// TwinCAT 3 PLC project Anker_Walfischgasse
// ProgramVersion: 3.1.4023.0
// libraries:
//   EfficientIO Communicator, * (EfficientIO)
//   EfficientIO Energy Basic, * (EfficientIO)
//   Lynus Persistent Data V1, * (Lynus AG)
//   Lynus Standards, * (EfficientIO)
//   Tc2_BABasic, * (Beckhoff Automation GmbH)
//   Tc2_Standard, * (Beckhoff Automation GmbH)
//   Tc2_System, * (Beckhoff Automation GmbH)
//   Tc2_Utilities, * (Beckhoff Automation GmbH)
//   Tc3_IotBase, * (Beckhoff Automation GmbH)
//   Tc3_JsonXml, * (Beckhoff Automation GmbH)
//   Tc3_Module, * (Beckhoff Automation GmbH)
// project tree:
//   / FastTask.TcTTO (not stored), MiddleTask.TcTTO, SlowTask.TcTTO (not stored)
//   FBs/ FB_Shelly_Pro1PM.TcPOU (not stored), FB_Shelly_Pro1PM_Helper.TcPOU, FB_TimeSwitch.TcPOU (not stored), FB_TimeSwitch_V2.TcPOU (not stored)
//   POUs/ prg5530Con.TcPOU, prg5530EMS.TcPOU, prgComEffIO.TcPOU, prg5530Grid.TcPOU (not stored), prgPersistent.TcPOU, prgRWEffIO.TcPOU (not stored), prgVarEffIO.TcPOU (not stored), prg_SystemTime.TcPOU (not stored)
// real-time tasks:
//   TASK FastTask: cycle T#5ms, priority 4, ADS port 350
//   TASK MiddleTask: cycle T#10ms, priority 8, ADS port 351
//   TASK SlowTask: cycle T#20ms, priority 10, ADS port 352
// I/O:
//   DEVICE Gerät 1 (Beckhoff CCAT)
//   DEVICE Gerät 2 (EtherCAT), AmsNetId 5.100.32.125.3.1
//     Klemme 1 (EK1200) [EK1200-5000 EtherCAT Netzteil (2A E-Bus)]
//       Klemme 2 (EL3443) [EL3443 3K. Leistungsmessung]
//       Klemme 3 (EL2652) [EL2652 2K. Relais Ausgang, Wechsler (230V AC / 30V DC)]
//       Klemme 4 (EL2652) [EL2652 2K. Relais Ausgang, Wechsler (230V AC / 30V DC)]
//       Klemme 5 (EL2652) [EL2652 2K. Relais Ausgang, Wechsler (230V AC / 30V DC)]
//       Klemme 6 (EL2652) [EL2652 2K. Relais Ausgang, Wechsler (230V AC / 30V DC)]
//       Klemme 7 (EL9011) [EL9011 Endklemme]

CONFIGURATION Anker_Walfischgasse
    RESOURCE PLC ON TwinCAT3
        TASK MiddleTask(INTERVAL := T#10ms, PRIORITY := 8);
        PROGRAM prgPersistent WITH MiddleTask : prgPersistent;
    END_RESOURCE
END_CONFIGURATION

// ---- POUs/prgPersistent.TcPOU
PROGRAM prgPersistent
VAR
	fbUSV		: FB_WritePersistentData_CX81xx;
	fb_Reboot		: NT_reboot;
	m_Reboot		: BOOL:=FALSE;
END_VAR

fbUSV(
	eSaveModeData:= eUSVSaveMode.eSaveWhenPowerfail, 
	bLoadPersistentDataOk=> , 
	bPowerFailDetect=> , 
	bError=> , 
	bySaveProcess=> , 
	dwStorageLast24h=> , 
	udiErrorCode=> );
	
prg_SystemTime();

		
fb_Reboot(	netid := '',
			delay := 2,
			start := m_Reboot);

END_PROGRAM

// ---- FBs/FB_Shelly_Pro1PM_Helper.TcPOU
FUNCTION_BLOCK FB_Shelly_Pro1PM_Helper
VAR_INPUT
	bSend			: BOOL;
	bSetOnP1		: BOOL;
	bSetOffP1		: BOOL;
END_VAR

VAR_IN_OUT
	fbClient		: FB_IotHttpClient;
END_VAR

VAR_OUTPUT
	bBusy			: BOOL;
	bError			: BOOL;
	bStateP1		: BOOL;
	lrapowerP1		: LREAL;
	lrvoltageP1		: LREAL;
	lraenergyP1		: LREAL;
	lrTemperatureP1	: LREAL;
END_VAR

VAR
	fbRequestSwitch0	: FB_IotHttpRequest;
	fbRequestSwitch1	: FB_IotHttpRequest;
	RisingEdge			: R_TRIG;
	RisingEdgeSetOnP1	: R_TRIG;
	RisingEdgeSetOffP1	: R_TRIG;
	fbJson				: FB_JsonDomParser;
	nState				: UDINT;
	timTimeout			: TON;
	tTimeOut			: TIME := T#2S;
	timTimeoutSwitch	: TON;
	tTimeOutSwitch		: TIME := T#5S;
	bGetContentResult	: BOOL;
	sContentS0			: STRING(511);
	
	bGetJsonResult		: BOOL;
	jsonDoc				: SJsonValue;
	jsonVal				: SJsonValue;
	
	nReqCount			: UDINT;	
	nResCount			: UDINT;
	nValidResCount		: UDINT;
	nErrCount			: UDINT;
	
	fbRequest2         : FB_IotHttpRequest;
	fbRequest3         : FB_IotHttpRequest;
	fbHeader            : FB_IotHttpHeaderFieldMap;
	fbHeader2            : FB_IotHttpHeaderFieldMap;
	
	sRealm	:	STRING(511);
	sPassword :	STRING(511) := ':sh3lly4ankerio2$$';
	snonce	:	STRING(511);
	scnonce	:	STRING(511);
	shash	: STRING(511);
	bhash	: BOOL;
	
	aData	: STRING(511);
	a_ha1	: ARRAY[0..31] OF BYTE;
	str_ha1 : STRING(511);
	str_Toha1   : STRING(511);
	udint_length_string : UDINT;
	
	a_ha2	: ARRAY[0..31] OF BYTE;
	str_ha2 : STRING(511);
	str_Toha2   : STRING(511);
	
	a_response	: ARRAY[0..31] OF BYTE;
	str_response : STRING(511);
	str_Toresponse   : STRING(511);

	str_authorization	: STRING(2048);
	
	sfincontent	: STRING(511);
	int_CountOffWrite: INT;
	int_CountOnWrite: INT;
	str_URI : STRING(50);
	int_Mode: INT;
	ton_Timeout: Ton;
	b_Done: BOOL;
	nState_Old: UDINT;
	int_ErrorCount: INT;
END_VAR

//Timer for Timeout
timTimeout(IN:= (nState = 1 AND bBusy) OR (nState = nState_Old AND bBusy), PT:= tTimeOut, Q=> , ET=> );
	IF timTimeout.Q THEN 
		nState := 0;
		bBusy := FALSE;
		bStateP1 := FALSE;
		lrapowerP1 := 0;
		lrvoltageP1 := 0;
		lraenergyP1 := 0;
		lrTemperatureP1 := 0;		
	END_IF
IF nState<> nState_old THEN
	nState_old := nState;
END_IF	
(*timTimeoutSwitch(IN:= bSetOnP1 OR bSetOffP1, PT:= tTimeOut, Q=> , ET=> );
	IF timTimeoutSwitch.Q THEN 
		bSetOnP1 := FALSE;
		bSetOffP1 := FALSE;
	END_IF
*)
IF bError THEN
	int_ErrorCount := int_ErrorCount+1;
	bError := FALSE;
END_IF

RisingEdge(CLK:= bSend );
RisingEdgeSetOnP1(CLK:= bSetOnP1 );
RisingEdgeSetOffP1(CLK:= bSetOffP1 );

CASE nState OF
	0:	
		IF RisingEdge.Q THEN 
			IF bSetOnP1 AND NOT b_Done THEN 
				// switch on
				str_URI :='/rpc/Switch.Set?id=0&on=true';
				int_Mode := 1;
				b_Done := TRUE;
				bBusy:= TRUE;
				bError:= FALSE;
				nState:= 1;
			ELSIF bSetOffP1 AND NOT b_Done THEN
				// switch off
				str_URI :='/rpc/Switch.Set?id=0&on=false';
				int_Mode := 2;
				b_Done := TRUE;
				bBusy:= TRUE;
				bError:= FALSE;
				nState:= 1;
			ELSIF ((bSetOnP1 OR bSetOffP1) AND  b_Done) OR (NOT bSetOnP1 AND NOT bSetOffP1) THEN
				// read
				str_URI :='/rpc/Switch.GetStatus?id=0';
				int_Mode := 0;
				b_Done := FALSE;
				bBusy:= TRUE;
				bError:= FALSE;
				nState:= 1;
			END_IF
		END_IF
	1:
		IF
			fbRequestSwitch0.SendRequest(sUri:=str_URI, fbClient:=fbClient, eRequestType:=ETcIotHttpRequestType.HTTP_Get, 0, 0, 0) THEN
			nState:= 2;
			nReqCount:= nReqCount+1;
		END_IF
	
	2:
		IF NOT fbRequestSwitch0.bBusy THEN
			bError:= TRUE;
			IF NOT fbRequestSwitch0.bError THEN
				bGetContentResult:= fbRequestSwitch0.GetHeaderField(pValue:= ADR(sContentS0), 
														 nValueSize:= SIZEOF(sContentS0), sField := 'WWW-Authenticate');
				IF fbRequestSwitch0.nStatusCode = 401 THEN
					bGetJsonResult:= FALSE;
						sRealm := sContentS0;
						sRealm := DELETE(sRealm, FIND(sRealm, 'realm') + 7, 0);
						sRealm := DELETE(sRealm, LEN(sRealm), FIND(sRealm, '"'));
						
						snonce := sContentS0;
						snonce := DELETE(snonce, FIND(snonce, 'nonce') + 7, 0);
						snonce := DELETE(snonce, LEN(snonce), FIND(snonce, '"'));
						
						scnonce := 'YmawvYzT';
					
						aData := sRealm;
						
						str_Toha1:=concat('admin:', sRealm);
						str_Toha1:=concat(str_Toha1, sPassword);
		 
						udint_length_string:= len2(ADR(str_Toha1));
						F_GenerateHashValue(E_HashMode.HASH_SHA256,ADR(str_Toha1),udint_length_string,ADR(a_ha1),32);
						
							str_ha1:=concat(byte_to_hexstr(a_ha1[0],2,TRUE),byte_to_hexstr(a_ha1[1],2,TRUE));
							str_ha1:=concat(str_ha1,byte_to_hexstr(a_ha1[2],2,TRUE));
							str_ha1:=concat(str_ha1,byte_to_hexstr(a_ha1[3],2,TRUE));
							str_ha1:=concat(str_ha1,byte_to_hexstr(a_ha1[4],2,TRUE));
							str_ha1:=concat(str_ha1,byte_to_hexstr(a_ha1[5],2,TRUE));
							str_ha1:=concat(str_ha1,byte_to_hexstr(a_ha1[6],2,TRUE));
							str_ha1:=concat(str_ha1,byte_to_hexstr(a_ha1[7],2,TRUE));
							str_ha1:=concat(str_ha1,byte_to_hexstr(a_ha1[8],2,TRUE));
							str_ha1:=concat(str_ha1,byte_to_hexstr(a_ha1[9],2,TRUE));
							str_ha1:=concat(str_ha1,byte_to_hexstr(a_ha1[10],2,TRUE));
							str_ha1:=concat(str_ha1,byte_to_hexstr(a_ha1[11],2,TRUE));
							str_ha1:=concat(str_ha1,byte_to_hexstr(a_ha1[12],2,TRUE));
							str_ha1:=concat(str_ha1,byte_to_hexstr(a_ha1[13],2,TRUE));
							str_ha1:=concat(str_ha1,byte_to_hexstr(a_ha1[14],2,TRUE));
							str_ha1:=concat(str_ha1,byte_to_hexstr(a_ha1[15],2,TRUE));
							str_ha1:=concat(str_ha1,byte_to_hexstr(a_ha1[16],2,TRUE));
							str_ha1:=concat(str_ha1,byte_to_hexstr(a_ha1[17],2,TRUE));
							str_ha1:=concat(str_ha1,byte_to_hexstr(a_ha1[18],2,TRUE));
							str_ha1:=concat(str_ha1,byte_to_hexstr(a_ha1[19],2,TRUE));
							str_ha1:=concat(str_ha1,byte_to_hexstr(a_ha1[20],2,TRUE));
							str_ha1:=concat(str_ha1,byte_to_hexstr(a_ha1[21],2,TRUE));
							str_ha1:=concat(str_ha1,byte_to_hexstr(a_ha1[22],2,TRUE));
							str_ha1:=concat(str_ha1,byte_to_hexstr(a_ha1[23],2,TRUE));
							str_ha1:=concat(str_ha1,byte_to_hexstr(a_ha1[24],2,TRUE));
							str_ha1:=concat(str_ha1,byte_to_hexstr(a_ha1[25],2,TRUE));
							str_ha1:=concat(str_ha1,byte_to_hexstr(a_ha1[26],2,TRUE));
							str_ha1:=concat(str_ha1,byte_to_hexstr(a_ha1[27],2,TRUE));
							str_ha1:=concat(str_ha1,byte_to_hexstr(a_ha1[28],2,TRUE));
							str_ha1:=concat(str_ha1,byte_to_hexstr(a_ha1[29],2,TRUE));
							str_ha1:=concat(str_ha1,byte_to_hexstr(a_ha1[30],2,TRUE));
							str_ha1:=concat(str_ha1,byte_to_hexstr(a_ha1[31],2,TRUE));
						
						str_Toha2:= concat('GET:',str_URI);
				 
						udint_length_string:= len2(ADR(str_Toha2));
						F_GenerateHashValue(E_HashMode.HASH_SHA256,ADR(str_Toha2),udint_length_string,ADR(a_ha2),32);
						
							str_ha2:=concat(byte_to_hexstr(a_ha2[0],2,TRUE),byte_to_hexstr(a_ha2[1],2,TRUE));
							str_ha2:=concat(str_ha2,byte_to_hexstr(a_ha2[2],2,TRUE));
							str_ha2:=concat(str_ha2,byte_to_hexstr(a_ha2[3],2,TRUE));
							str_ha2:=concat(str_ha2,byte_to_hexstr(a_ha2[4],2,TRUE));
							str_ha2:=concat(str_ha2,byte_to_hexstr(a_ha2[5],2,TRUE));
							str_ha2:=concat(str_ha2,byte_to_hexstr(a_ha2[6],2,TRUE));
							str_ha2:=concat(str_ha2,byte_to_hexstr(a_ha2[7],2,TRUE));
							str_ha2:=concat(str_ha2,byte_to_hexstr(a_ha2[8],2,TRUE));
							str_ha2:=concat(str_ha2,byte_to_hexstr(a_ha2[9],2,TRUE));
							str_ha2:=concat(str_ha2,byte_to_hexstr(a_ha2[10],2,TRUE));
							str_ha2:=concat(str_ha2,byte_to_hexstr(a_ha2[11],2,TRUE));
							str_ha2:=concat(str_ha2,byte_to_hexstr(a_ha2[12],2,TRUE));
							str_ha2:=concat(str_ha2,byte_to_hexstr(a_ha2[13],2,TRUE));
							str_ha2:=concat(str_ha2,byte_to_hexstr(a_ha2[14],2,TRUE));
							str_ha2:=concat(str_ha2,byte_to_hexstr(a_ha2[15],2,TRUE));
							str_ha2:=concat(str_ha2,byte_to_hexstr(a_ha2[16],2,TRUE));
							str_ha2:=concat(str_ha2,byte_to_hexstr(a_ha2[17],2,TRUE));
							str_ha2:=concat(str_ha2,byte_to_hexstr(a_ha2[18],2,TRUE));
							str_ha2:=concat(str_ha2,byte_to_hexstr(a_ha2[19],2,TRUE));
							str_ha2:=concat(str_ha2,byte_to_hexstr(a_ha2[20],2,TRUE));
							str_ha2:=concat(str_ha2,byte_to_hexstr(a_ha2[21],2,TRUE));
							str_ha2:=concat(str_ha2,byte_to_hexstr(a_ha2[22],2,TRUE));
							str_ha2:=concat(str_ha2,byte_to_hexstr(a_ha2[23],2,TRUE));
							str_ha2:=concat(str_ha2,byte_to_hexstr(a_ha2[24],2,TRUE));
							str_ha2:=concat(str_ha2,byte_to_hexstr(a_ha2[25],2,TRUE));
							str_ha2:=concat(str_ha2,byte_to_hexstr(a_ha2[26],2,TRUE));
							str_ha2:=concat(str_ha2,byte_to_hexstr(a_ha2[27],2,TRUE));
							str_ha2:=concat(str_ha2,byte_to_hexstr(a_ha2[28],2,TRUE));
							str_ha2:=concat(str_ha2,byte_to_hexstr(a_ha2[29],2,TRUE));
							str_ha2:=concat(str_ha2,byte_to_hexstr(a_ha2[30],2,TRUE));
							str_ha2:=concat(str_ha2,byte_to_hexstr(a_ha2[31],2,TRUE));
							
						// <ha1> + ":" + <nonce> + ":" + <nc> + ":" + <cnonce> + ":" + "auth" + ":" + <ha2>
						
						str_Toresponse:=concat(str_ha1,':');
						str_Toresponse:=concat(str_Toresponse,snonce);
						str_Toresponse:=concat(str_Toresponse,':00000001:');
						str_Toresponse:=concat(str_Toresponse,scnonce);
						str_Toresponse:=concat(str_Toresponse,':');
						str_Toresponse:=concat(str_Toresponse,'auth:');
						str_Toresponse:=concat(str_Toresponse,str_ha2);
						
						udint_length_string:= len2(ADR(str_Toresponse));
						F_GenerateHashValue(E_HashMode.HASH_SHA256,ADR(str_Toresponse),udint_length_string,ADR(a_response),32);
						
							str_response:=concat(byte_to_hexstr(a_response[0],2,TRUE),byte_to_hexstr(a_response[1],2,TRUE));
							str_response:=concat(str_response,byte_to_hexstr(a_response[2],2,TRUE));
							str_response:=concat(str_response,byte_to_hexstr(a_response[3],2,TRUE));
							str_response:=concat(str_response,byte_to_hexstr(a_response[4],2,TRUE));
							str_response:=concat(str_response,byte_to_hexstr(a_response[5],2,TRUE));
							str_response:=concat(str_response,byte_to_hexstr(a_response[6],2,TRUE));
							str_response:=concat(str_response,byte_to_hexstr(a_response[7],2,TRUE));
							str_response:=concat(str_response,byte_to_hexstr(a_response[8],2,TRUE));
							str_response:=concat(str_response,byte_to_hexstr(a_response[9],2,TRUE));
							str_response:=concat(str_response,byte_to_hexstr(a_response[10],2,TRUE));
							str_response:=concat(str_response,byte_to_hexstr(a_response[11],2,TRUE));
							str_response:=concat(str_response,byte_to_hexstr(a_response[12],2,TRUE));
							str_response:=concat(str_response,byte_to_hexstr(a_response[13],2,TRUE));
							str_response:=concat(str_response,byte_to_hexstr(a_response[14],2,TRUE));
							str_response:=concat(str_response,byte_to_hexstr(a_response[15],2,TRUE));
							str_response:=concat(str_response,byte_to_hexstr(a_response[16],2,TRUE));
							str_response:=concat(str_response,byte_to_hexstr(a_response[17],2,TRUE));
							str_response:=concat(str_response,byte_to_hexstr(a_response[18],2,TRUE));
							str_response:=concat(str_response,byte_to_hexstr(a_response[19],2,TRUE));
							str_response:=concat(str_response,byte_to_hexstr(a_response[20],2,TRUE));
							str_response:=concat(str_response,byte_to_hexstr(a_response[21],2,TRUE));
							str_response:=concat(str_response,byte_to_hexstr(a_response[22],2,TRUE));
							str_response:=concat(str_response,byte_to_hexstr(a_response[23],2,TRUE));
							str_response:=concat(str_response,byte_to_hexstr(a_response[24],2,TRUE));
							str_response:=concat(str_response,byte_to_hexstr(a_response[25],2,TRUE));
							str_response:=concat(str_response,byte_to_hexstr(a_response[26],2,TRUE));
							str_response:=concat(str_response,byte_to_hexstr(a_response[27],2,TRUE));
							str_response:=concat(str_response,byte_to_hexstr(a_response[28],2,TRUE));
							str_response:=concat(str_response,byte_to_hexstr(a_response[29],2,TRUE));
							str_response:=concat(str_response,byte_to_hexstr(a_response[30],2,TRUE));
							str_response:=concat(str_response,byte_to_hexstr(a_response[31],2,TRUE));
							
						// "Digest username=\"admin\", realm=\"shellypro4pm-083af27cfbac\", nonce=\"63768368\", uri=\"/rpc/Switch.GetStatus?id=0\", algorithm=\"SHA-256\", qop=auth, nc=00000001, cnonce=\"oKOklSrS\", response=\"d1d59d1e015dee0a3acfc97b20a0fa0ff851b03d79ca00df59ce018a63041468\""
						
						str_authorization:=concat('Digest username="admin", realm="',sRealm);
						str_authorization:=concat(str_authorization,'", nonce="');
						str_authorization:=concat(str_authorization,snonce);
						str_authorization:=concat(str_authorization,'", algorithm="SHA-256", uri="');
						str_authorization:=concat(str_authorization,str_URI);
						str_authorization:=concat(str_authorization,'", qop=auth, nc=00000001, cnonce="');
						str_authorization:=concat(str_authorization,scnonce);
						str_authorization:=concat(str_authorization,'", response="');
						str_authorization:=concat(str_authorization,str_response);
						str_authorization:=concat(str_authorization,'"');
						
						fbHeader.AddField('Authorization', str_authorization, FALSE);
						IF fbRequest2.SendRequest(sUri:= str_URI, fbClient:= fbClient, eRequestType:= ETcIotHttpRequestType.HTTP_Get, 0, 0, fbHeader) THEN
							nState:= 3;
							bBusy:= TRUE;
							bError:= FALSE;
						END_IF
				END_IF
			END_IF
		END_IF
	
	3:
		IF NOT fbRequest2.bBusy THEN
			bError:= TRUE;
			IF int_Mode<>0 THEN
				bError:= FALSE;
			END_IF
			IF NOT fbRequest2.bError THEN		//AND int_Mode=0 				 
				bGetContentResult:= fbRequest2.GetContent(pContent:= ADR(sfincontent), nContentSize:= SIZEOF(sfincontent), bSetNullTermination:= TRUE);
	
				IF fbRequest2.nStatusCode >= 200 AND fbRequest2.nStatusCode < 300 THEN
					bGetJsonResult:= FALSE;
					jsonDoc:= fbRequest2.GetJsonDomContent(fbJson);
					IF jsonDoc <> 0 THEN
						bGetJsonResult:= TRUE;
						IF fbJson.HasMember(jsonDoc, 'output')  THEN
							jsonVal:= fbJson.FindMember(jsonDoc, 'output');
							nValidResCount:= nValidResCount+1;					
							IF fbJson.IsBool(jsonVal) AND (fbJson.GetBool(jsonVal)=TRUE OR fbJson.GetBool(jsonVal)=FALSE) THEN							
								bStateP1:= fbJson.GetBool(jsonVal);									
							END_IF
						END_IF
						IF fbJson.HasMember(jsonDoc, 'apower')  THEN
							jsonVal:= fbJson.FindMember(jsonDoc, 'apower');
							nValidResCount:= nValidResCount+1;
							IF fbJson.IsDouble(jsonVal) AND fbJson.GetDouble(jsonVal)> -3.402823E+38 AND fbJson.GetDouble(jsonVal)< 3.402823E+38 THEN							
								lrapowerP1:= fbJson.GetDouble(jsonVal);									
							END_IF
						END_IF
						IF fbJson.HasMember(jsonDoc, 'voltage')  THEN
							jsonVal:= fbJson.FindMember(jsonDoc, 'voltage');
							nValidResCount:= nValidResCount+1;					
							IF fbJson.IsDouble(jsonVal) AND fbJson.GetDouble(jsonVal)> -3.402823E+38 AND fbJson.GetDouble(jsonVal)< 3.402823E+38 THEN
								lrvoltageP1:= fbJson.GetDouble(jsonVal);									
							END_IF
						END_IF
						IF fbJson.HasMember(jsonDoc, 'temperature')  THEN
							jsonVal:= fbJson.FindMember(jsonDoc, 'temperature');
							 IF fbJson.HasMember(jsonVal, 'tC') AND fbJson.GetDouble(jsonVal)> -3.402823E+38 AND fbJson.GetDouble(jsonVal)< 3.402823E+38 THEN							
								jsonVal:= fbJson.FindMember(jsonVal, 'tC');
								nValidResCount:= nValidResCount+1;					
								IF fbJson.IsDouble(jsonVal) AND fbJson.GetDouble(jsonVal)> -3.402823E+38 AND fbJson.GetDouble(jsonVal)< 3.402823E+38 THEN
									lrTemperatureP1:= fbJson.GetDouble(jsonVal);									
								END_IF
							END_IF
						END_IF
						IF fbJson.HasMember(jsonDoc, 'aenergy')  THEN
							jsonVal:= fbJson.FindMember(jsonDoc, 'aenergy');
							IF fbJson.HasMember(jsonVal, 'total') AND fbJson.GetDouble(jsonVal)> -3.402823E+38 AND fbJson.GetDouble(jsonVal)< 3.402823E+38 THEN							
								jsonVal:= fbJson.FindMember(jsonVal, 'total');
								nValidResCount:= nValidResCount+1;
								IF fbJson.IsDouble(jsonVal) AND fbJson.GetDouble(jsonVal)> -3.402823E+38 AND fbJson.GetDouble(jsonVal)< 3.402823E+38 THEN
									lraenergyP1:= fbJson.GetDouble(jsonVal);
								END_IF
							bError:= FALSE;
							END_IF
						END_IF	
					nResCount:= nResCount+1;			
					END_IF
				END_IF
			END_IF
		nState:= 4;
//		bBusy:= FALSE;
			IF bError THEN
				nErrCount:= nErrCount+1;
			END_IF
		ELSE
			ton_Timeout.IN := TRUE;
			IF ton_Timeout.Q THEN
				nState:= 3;	
				ton_Timeout.IN := FALSE;
			END_IF
		END_IF
	
	
	4:
		ton_Timeout.IN := FALSE;
		nState:= 6;
		
	6:
		bBusy:= FALSE;
		nState:= 0;

	
END_CASE

ton_Timeout(PT := T#5S);

END_FUNCTION_BLOCK

// ---- POUs/prg5530Con.TcPOU
PROGRAM prg5530Con
VAR
	// Shelly1: 
	lrS1P1Power				:	LREAL;			//{#lynus.ag#()}
	lrS1P1Power_kW			:	LREAL;			//{#lynus.ag#()}
	lrS1P1Voltage			:	LREAL;			//{#lynus.ag#()}
	lrS1P1Energy			:	LREAL;			//{#lynus.ag#()}
	lrS1P1Temperature		:	LREAL;			//{#lynus.ag#()}
	bS1P1On					:	BOOL;			//{#lynus.ag#()}
	bS1P1Off				:	BOOL;			//{#lynus.ag#()}
	bS1P1Switch				:	BOOL;			//{#lynus.ag#()}
	
	// Shelly2: 
//	fbShelly2				:	FB_Shelly_Pro1PM;
	lrS2P1Power				:	LREAL;			//{#lynus.ag#()}
	lrS2P1Power_kW			:	LREAL;			//{#lynus.ag#()}
	lrS2P1Voltage			:	LREAL;			//{#lynus.ag#()}
	lrS2P1Energy			:	LREAL;			//{#lynus.ag#()}
	lrS2P1Temperature		:	LREAL;			//{#lynus.ag#()}
	bS2P1On					:	BOOL;			//{#lynus.ag#()}
	bS2P1Off				:	BOOL;			//{#lynus.ag#()}
	bS2P1Switch				:	BOOL;			//{#lynus.ag#()}
	
	// Shelly3: 
//	fbShelly3				:	FB_Shelly_Pro1PM;
	lrS3P1Power				:	LREAL;			//{#lynus.ag#()}
	lrS3P1Power_kW			:	LREAL;			//{#lynus.ag#()}
	lrS3P1Voltage			:	LREAL;			//{#lynus.ag#()}
	lrS3P1Energy			:	LREAL;			//{#lynus.ag#()}
	lrS3P1Temperature		:	LREAL;			//{#lynus.ag#()}
	bS3P1On					:	BOOL;			//{#lynus.ag#()}
	bS3P1Off				:	BOOL;			//{#lynus.ag#()}
	bS3P1Switch				:	BOOL;			//{#lynus.ag#()}
	
	// Shelly4: 
//	fbShelly4				:	FB_Shelly_Pro1PM;
	lrS4P1Power				:	LREAL;			//{#lynus.ag#()}
	lrS4P1Power_kW			:	LREAL;			//{#lynus.ag#()}
	lrS4P1Voltage			:	LREAL;			//{#lynus.ag#()}
	lrS4P1Energy			:	LREAL;			//{#lynus.ag#()}
	lrS4P1Temperature		:	LREAL;			//{#lynus.ag#()}
	bS4P1On					:	BOOL;			//{#lynus.ag#()}
	bS4P1Off				:	BOOL;			//{#lynus.ag#()}
	bS4P1Switch				:	BOOL;			//{#lynus.ag#()}
	
	// Shelly5: 
//	fbShelly5				:	FB_Shelly_Pro1PM;
	lrS5P1Power				:	LREAL;			//{#lynus.ag#()}
	lrS5P1Power_kW			:	LREAL;			//{#lynus.ag#()}
	lrS5P1Voltage			:	LREAL;			//{#lynus.ag#()}
	lrS5P1Energy			:	LREAL;			//{#lynus.ag#()}
	lrS5P1Temperature		:	LREAL;			//{#lynus.ag#()}
	bS5P1On					:	BOOL;			//{#lynus.ag#()}
	bS5P1Off				:	BOOL;			//{#lynus.ag#()}
	bS5P1Switch				:	BOOL;			//{#lynus.ag#()}
	
	// Shelly6: 
	lrS6P1Power				:	LREAL;			//{#lynus.ag#()}
	lrS6P1Power_kW			:	LREAL;			//{#lynus.ag#()}
	lrS6P1Voltage			:	LREAL;			//{#lynus.ag#()}
	lrS6P1Energy			:	LREAL;			//{#lynus.ag#()}
	lrS6P1Temperature		:	LREAL;			//{#lynus.ag#()}
	bS6P1On					:	BOOL;			//{#lynus.ag#()}
	bS6P1Off				:	BOOL;			//{#lynus.ag#()}
	bS6P1Switch				:	BOOL;			//{#lynus.ag#()}
	
	// Shelly7: 
	lrS7P1Power				:	LREAL;			//{#lynus.ag#()}
	lrS7P1Power_kW			:	LREAL;			//{#lynus.ag#()}
	lrS7P1Voltage			:	LREAL;			//{#lynus.ag#()}
	lrS7P1Energy			:	LREAL;			//{#lynus.ag#()}
	lrS7P1Temperature		:	LREAL;			//{#lynus.ag#()}
	bS7P1On					:	BOOL;			//{#lynus.ag#()}
	bS7P1Off				:	BOOL;			//{#lynus.ag#()}
	bS7P1Switch				:	BOOL;			//{#lynus.ag#()}
	
	// Shelly8: 
	lrS8P1Power				:	LREAL;			//{#lynus.ag#()}
	lrS8P1Power_kW			:	LREAL;			//{#lynus.ag#()}
	lrS8P1Voltage			:	LREAL;			//{#lynus.ag#()}
	lrS8P1Energy			:	LREAL;			//{#lynus.ag#()}
	lrS8P1Temperature		:	LREAL;			//{#lynus.ag#()}
	bS8P1On					:	BOOL;			//{#lynus.ag#()}
	bS8P1Off				:	BOOL;			//{#lynus.ag#()}
	bS8P1Switch				:	BOOL;			//{#lynus.ag#()}
	
	// Shelly9: 
	lrS9P1Power				:	LREAL;			//{#lynus.ag#()}
	lrS9P1Power_kW			:	LREAL;			//{#lynus.ag#()}
	lrS9P1Voltage			:	LREAL;			//{#lynus.ag#()}
	lrS9P1Energy			:	LREAL;			//{#lynus.ag#()}
	lrS9P1Temperature		:	LREAL;			//{#lynus.ag#()}
	bS9P1On					:	BOOL;			//{#lynus.ag#()}
	bS9P1Off				:	BOOL;			//{#lynus.ag#()}
	bS9P1Switch				:	BOOL;			//{#lynus.ag#()}
	
	// Shelly10: 
	lrS10P1Power			:	LREAL;			//{#lynus.ag#()}
	lrS10P1Power_kW 		:	LREAL;			//{#lynus.ag#()}
	lrS10P1Voltage			:	LREAL;			//{#lynus.ag#()}
	lrS10P1Energy			:	LREAL;			//{#lynus.ag#()}
	lrS10P1Temperature		:	LREAL;			//{#lynus.ag#()}
	bS10P1On				:	BOOL;			//{#lynus.ag#()}
	bS10P1Off				:	BOOL;			//{#lynus.ag#()}
	bS10P1Switch			:	BOOL;			//{#lynus.ag#()}
	
	// Shelly11: 
	lrS11P1Power			:	LREAL;			//{#lynus.ag#()}
	lrS11P1Power_kW			:	LREAL;			//{#lynus.ag#()}
	lrS11P1Voltage			:	LREAL;			//{#lynus.ag#()}
	lrS11P1Energy			:	LREAL;			//{#lynus.ag#()}
	lrS11P1Temperature		:	LREAL;			//{#lynus.ag#()}
	bS11P1On				:	BOOL;			//{#lynus.ag#()}
	bS11P1Off				:	BOOL;			//{#lynus.ag#()}
	bS11P1Switch			:	BOOL;			//{#lynus.ag#()}
	
	// Shelly12: 
	lrS12P1Power			:	LREAL;			//{#lynus.ag#()}
	lrS12P1Power_kW			:	LREAL;			//{#lynus.ag#()}
	lrS12P1Voltage			:	LREAL;			//{#lynus.ag#()}
	lrS12P1Energy			:	LREAL;			//{#lynus.ag#()}
	lrS12P1Temperature		:	LREAL;			//{#lynus.ag#()}
	bS12P1On				:	BOOL;			//{#lynus.ag#()}
	bS12P1Off				:	BOOL;			//{#lynus.ag#()}
	bS12P1Switch			:	BOOL;			//{#lynus.ag#()}
	
	// Shelly13: 
	lrS13P1Power			:	LREAL;			//{#lynus.ag#()}
	lrS13P1Power_kW			:	LREAL;			//{#lynus.ag#()}
	lrS13P1Voltage			:	LREAL;			//{#lynus.ag#()}
	lrS13P1Energy			:	LREAL;			//{#lynus.ag#()}
	lrS13P1Temperature		:	LREAL;			//{#lynus.ag#()}
	bS13P1On				:	BOOL;			//{#lynus.ag#()}
	bS13P1Off				:	BOOL;			//{#lynus.ag#()}
	bS13P1Switch			:	BOOL;			//{#lynus.ag#()}
	
	// Shelly14: 
	lrS14P1Power			:	LREAL;			//{#lynus.ag#()}
	lrS14P1Power_kW			:	LREAL;			//{#lynus.ag#()}
	lrS14P1Voltage			:	LREAL;			//{#lynus.ag#()}
	lrS14P1Energy			:	LREAL;			//{#lynus.ag#()}
	lrS14P1Temperature		:	LREAL;			//{#lynus.ag#()}
	bS14P1On				:	BOOL;			//{#lynus.ag#()}
	bS14P1Off				:	BOOL;			//{#lynus.ag#()}
	bS14P1Switch			:	BOOL;			//{#lynus.ag#()}
	
	// Other
	lrRemainPower_kW		:	LREAL;			//{#lynus.ag#()}
	
	// state maschine for GET requests
	str_Array_IPs			: array[1..30] of STRING(15);			//arrays for IPs
	int_State: INT;													// state
	
	// Shelly: 
	ton_TimeOut: Ton;
	int_Multiplier_1 			:INT:=1;								// multilpier received values, =2 when external fuse is on, was at the beginning
	int_Multiplier_2 			:INT:=1;								// multilpier received values, =2 when external fuse is on, was at the beginning
	int_Multiplier_3 			:INT:=1;								// multilpier received values, =2 when external fuse is on, was at the beginning
	int_Multiplier_4 			:INT:=1;								// multilpier received values, =2 when external fuse is on, was at the beginning
	int_Multiplier_5 			:INT:=1;								// multilpier received values, =2 when external fuse is on, was at the beginning
	int_Multiplier_6 			:INT:=1;								// multilpier received values, =2 when external fuse is on, was at the beginning
	int_Multiplier_7 			:INT:=1;								// multilpier received values, =2 when external fuse is on, was at the beginning
	int_Multiplier_8 			:INT:=1;								// multilpier received values, =2 when external fuse is on, was at the beginning
	int_Multiplier_9 			:INT:=1;								// multilpier received values, =2 when external fuse is on, was at the beginning
	int_Multiplier_10 			:INT:=1;								// multilpier received values, =2 when external fuse is on, was at the beginning
	int_Multiplier_11 			:INT:=1;								// multilpier received values, =2 when external fuse is on, was at the beginning
	int_Multiplier_12 			:INT:=1;								// multilpier received values, =2 when external fuse is on, was at the beginning
	int_Multiplier_13 			:INT:=1;								// multilpier received values, =2 when external fuse is on, was at the beginning
	int_Multiplier_14 			:INT:=1;								// multilpier received values, =2 when external fuse is on, was at the beginning

	int_TimeoutCounter: ARRAY[1..30] OF INT;	
	int_SuccessCounter: ARRAY[1..30] OF INT;	
	int_ErrorCounter: ARRAY[1..30] OF INT;
	ton_wait: Ton;
	fbShelly				:	ARRAY[1..20] OF FB_Shelly_Pro1PM;
	f_Trig_Busy				:	ARRAY[1..20] OF f_trig;
	m_Error_HTTP: BOOL;							//{#lynus.ag#()}
	m_Start: BOOL;
END_VAR

CASE int_State OF
	0: 		// Init State
	
	// define IPs
	str_Array_IPs[1]	:='10.55.30.131';
	str_Array_IPs[2]	:='10.55.30.132';
	str_Array_IPs[3]	:='10.55.30.133';
	str_Array_IPs[4]	:='10.55.30.134';
	str_Array_IPs[5]	:='10.55.30.135';
	str_Array_IPs[6]	:='10.55.30.136';
	str_Array_IPs[7]	:='10.55.30.137';
	str_Array_IPs[8]	:='10.55.30.138';
	str_Array_IPs[9]	:='10.55.30.139';
	str_Array_IPs[10]	:='10.55.30.140';
	str_Array_IPs[11]	:='10.55.30.141';
	str_Array_IPs[12]	:='10.55.30.142';
	str_Array_IPs[13]	:='10.55.30.143';
	str_Array_IPs[14]	:='10.55.30.144';
	
	// =2 for the beginning when bypass fuse is on
	int_Multiplier_1 		:=2;
	int_Multiplier_2 		:=2;	
	int_Multiplier_3 		:=2;
	int_Multiplier_4 		:=1;
	int_Multiplier_5 		:=1;
	int_Multiplier_6 		:=1;
	int_Multiplier_7 		:=1;
	int_Multiplier_8 		:=2;
	int_Multiplier_9 		:=2;
	int_Multiplier_10 		:=2;
	int_Multiplier_11 		:=1;
	int_Multiplier_12 		:=1;
	int_Multiplier_13 		:=1;	
	int_Multiplier_14 		:=1;	

	IF str_Array_IPs[1] <> '' THEN
		int_State :=1;
	END_IF
		
	1: 		// request
	
	fbShelly[int_State].bStart		:= TRUE;
	fbShelly[int_State].sHostname	:= str_Array_IPs[int_State];

	// values to transfer to shelly
	fbShelly[int_State].bOnP1		:= bS1P1On;
	fbShelly[int_State].bOffP1		:= bS1P1Off;
	
	ton_TimeOut.IN 		:= TRUE;
	f_Trig_Busy[int_State](clk	:= fbShelly[int_State].bBusy);

	IF  ton_TimeOut.Q THEN		// timeout
		int_TimeoutCounter[int_State]	:= int_TimeoutCounter[int_State]+1;
		fbShelly[int_State].bStart		:= FALSE;
		ton_TimeOut.IN 		:= FALSE;
		// go to next state
		IF 	int_state < 30 AND str_Array_IPs[int_State+1] <> '' THEN	
			int_State := int_State+1;
		ELSE
			int_State := 100;			// wait state for new run
		END_IF		
	ELSIF  fbShelly[int_State].bError THEN		// error
		int_ErrorCounter[int_State]	:= int_ErrorCounter[int_State]+1;
		fbShelly[int_State].bStart		:= FALSE;
		ton_TimeOut.IN 		:= FALSE;
		// go to next state
		IF 	int_state < 30 AND str_Array_IPs[int_State+1] <> '' THEN	
			int_State := int_State+1;
		ELSE
			int_State := 100;			// wait state for new run
		END_IF	
	ELSIF f_Trig_Busy[int_State].Q AND NOT fbShelly[int_State].bError AND NOT ton_TimeOut.Q THEN		// received values
		int_SuccessCounter[int_State]	:= int_SuccessCounter[int_State]+1;
		fbShelly[int_State].bStart		:= FALSE;
		ton_TimeOut.IN 		:= FALSE;
	
		
		// copy received values
		lrS1P1Voltage	:= fbShelly[int_State].lrvoltageP1; 
		lrS1P1Power 	:= fbShelly[int_State].lrpowerP1 * int_Multiplier_1;
		lrS1P1Energy 	:= fbShelly[int_State].lrenergyP1 *int_Multiplier_1;
		lrS1P1Temperature :=fbShelly[int_State].lrTemperatureP1;
		bS1P1Switch		:= fbShelly[int_State].bStateP1;
		
		// go to next state
		IF 	int_state < 30 AND str_Array_IPs[int_State+1] <> '' THEN	
			int_State :=int_State+1;
		ELSE
			int_State := 100;			// wait state for new run
		END_IF
	END_IF
	
	2: 		// request
	
	fbShelly[int_State].bStart		:= TRUE;
	fbShelly[int_State].sHostname	:= str_Array_IPs[int_State];

	// values to transfer to shelly
	fbShelly[int_State].bOnP1		:= bS2P1On;
	fbShelly[int_State].bOffP1		:= bS2P1Off;
	
	ton_TimeOut.IN 		:= TRUE;
	f_Trig_Busy[int_State](clk	:= fbShelly[int_State].bBusy);

	IF  ton_TimeOut.Q THEN		// timeout
		int_TimeoutCounter[int_State]	:= int_TimeoutCounter[int_State]+1;
		fbShelly[int_State].bStart		:= FALSE;
		ton_TimeOut.IN 		:= FALSE;
		// go to next state
		IF 	int_state < 30 AND str_Array_IPs[int_State+1] <> '' THEN	
			int_State := int_State+1;
		ELSE
			int_State := 100;			// wait state for new run
		END_IF		
	ELSIF  fbShelly[int_State].bError THEN		// error
		int_ErrorCounter[int_State]	:= int_ErrorCounter[int_State]+1;
		fbShelly[int_State].bStart		:= FALSE;
		ton_TimeOut.IN 		:= FALSE;
		// go to next state
		IF 	int_state < 30 AND str_Array_IPs[int_State+1] <> '' THEN	
			int_State := int_State+1;
		ELSE
			int_State := 100;			// wait state for new run
		END_IF	
	ELSIF f_Trig_Busy[int_State].Q AND NOT fbShelly[int_State].bError AND NOT ton_TimeOut.Q THEN		// received values
		int_SuccessCounter[int_State]	:= int_SuccessCounter[int_State]+1;
		fbShelly[int_State].bStart		:= FALSE;
		ton_TimeOut.IN 		:= FALSE;
	
		
		// copy received values
		lrS2P1Voltage	:= fbShelly[int_State].lrvoltageP1; 
		lrS2P1Power 	:= fbShelly[int_State].lrpowerP1 * int_Multiplier_2;
		lrS2P1Energy 	:= fbShelly[int_State].lrenergyP1 *int_Multiplier_2;
		lrS2P1Temperature :=fbShelly[int_State].lrTemperatureP1;
		bS2P1Switch		:= fbShelly[int_State].bStateP1;
	

		// go to next state
		IF 	int_state < 30 AND str_Array_IPs[int_State+1] <> '' THEN	
			int_State :=int_State+1;
		ELSE
			int_State := 100;			// wait state for new run
		END_IF
	END_IF

	3: 		// request
	
	fbShelly[int_State].bStart		:= TRUE;
	fbShelly[int_State].sHostname	:= str_Array_IPs[int_State];

	// values to transfer to shelly
	fbShelly[int_State].bOnP1		:= bS3P1On;
	fbShelly[int_State].bOffP1		:= bS3P1Off;
	
	ton_TimeOut.IN 		:= TRUE;
	f_Trig_Busy[int_State] (clk	:= fbShelly[int_State].bBusy);

	IF  ton_TimeOut.Q THEN		// timeout
		int_TimeoutCounter[int_State]	:= int_TimeoutCounter[int_State]+1;
		fbShelly[int_State].bStart		:= FALSE;
		ton_TimeOut.IN 		:= FALSE;
		// go to next state
		IF 	int_state < 30 AND str_Array_IPs[int_State+1] <> '' THEN	
			int_State := int_State+1;
		ELSE
			int_State := 100;			// wait state for new run
		END_IF		
	ELSIF  fbShelly[int_State].bError THEN		// error
		int_ErrorCounter[int_State]	:= int_ErrorCounter[int_State]+1;
		fbShelly[int_State].bStart		:= FALSE;
		ton_TimeOut.IN 		:= FALSE;
		// go to next state
		IF 	int_state < 30 AND str_Array_IPs[int_State+1] <> '' THEN	
			int_State := int_State+1;
		ELSE
			int_State := 100;			// wait state for new run
		END_IF	
	ELSIF f_Trig_Busy[int_State].Q AND NOT fbShelly[int_State].bError AND NOT ton_TimeOut.Q THEN		// received values
		int_SuccessCounter[int_State]	:= int_SuccessCounter[int_State]+1;
		fbShelly[int_State].bStart		:= FALSE;
		ton_TimeOut.IN 		:= FALSE;
	
		
		// copy received values
		lrS3P1Voltage	:= fbShelly[int_State].lrvoltageP1; 
		lrS3P1Power 	:= fbShelly[int_State].lrpowerP1 * int_Multiplier_3;
		lrS3P1Energy 	:= fbShelly[int_State].lrenergyP1 *int_Multiplier_3;
		lrS3P1Temperature :=fbShelly[int_State].lrTemperatureP1;
		bS3P1Switch		:= fbShelly[int_State].bStateP1;
	

		// go to next state
		IF 	int_state < 30 AND str_Array_IPs[int_State+1] <> '' THEN	
			int_State :=int_State+1;
		ELSE
			int_State := 100;			// wait state for new run
		END_IF
	END_IF	
	
	4: 		// request
	
	fbShelly[int_State].bStart		:= TRUE;
	fbShelly[int_State].sHostname	:= str_Array_IPs[int_State];

	// values to transfer to shelly
	fbShelly[int_State].bOnP1		:= bS4P1On;
	fbShelly[int_State].bOffP1		:= bS4P1Off;
	
	ton_TimeOut.IN 		:= TRUE;
	f_Trig_Busy[int_State] (clk	:= fbShelly[int_State].bBusy);

	IF  ton_TimeOut.Q THEN		// timeout
		int_TimeoutCounter[int_State]	:= int_TimeoutCounter[int_State]+1;
		fbShelly[int_State].bStart		:= FALSE;
		ton_TimeOut.IN 		:= FALSE;
		// go to next state
		IF 	int_state < 30 AND str_Array_IPs[int_State+1] <> '' THEN	
			int_State := int_State+1;
		ELSE
			int_State := 100;			// wait state for new run
		END_IF		
	ELSIF  fbShelly[int_State].bError THEN		// error
		int_ErrorCounter[int_State]	:= int_ErrorCounter[int_State]+1;
		fbShelly[int_State].bStart		:= FALSE;
		ton_TimeOut.IN 		:= FALSE;
		// go to next state
		IF 	int_state < 30 AND str_Array_IPs[int_State+1] <> '' THEN	
			int_State := int_State+1;
		ELSE
			int_State := 100;			// wait state for new run
		END_IF	
	ELSIF f_Trig_Busy[int_State].Q AND NOT fbShelly[int_State].bError AND NOT ton_TimeOut.Q THEN		// received values
		int_SuccessCounter[int_State]	:= int_SuccessCounter[int_State]+1;
		fbShelly[int_State].bStart		:= FALSE;
		ton_TimeOut.IN 		:= FALSE;
	
		
		// copy received values
		lrS4P1Voltage	:= fbShelly[int_State].lrvoltageP1; 
		lrS4P1Power 	:= fbShelly[int_State].lrpowerP1 * int_Multiplier_4;
		lrS4P1Energy 	:= fbShelly[int_State].lrenergyP1 *int_Multiplier_4;
		lrS4P1Temperature :=fbShelly[int_State].lrTemperatureP1;
		bS4P1Switch		:= fbShelly[int_State].bStateP1;
	

		// go to next state
		IF 	int_state < 30 AND str_Array_IPs[int_State+1] <> '' THEN	
			int_State :=int_State+1;
		ELSE
			int_State := 100;			// wait state for new run
		END_IF
	END_IF		
	
	5: 		// request
	
	fbShelly[int_State].bStart		:= TRUE;
	fbShelly[int_State].sHostname	:= str_Array_IPs[int_State];

	// values to transfer to shelly
	fbShelly[int_State].bOnP1		:= bS5P1On;
	fbShelly[int_State].bOffP1		:= bS5P1Off;
	
	ton_TimeOut.IN 		:= TRUE;
	f_Trig_Busy[int_State] (clk	:= fbShelly[int_State].bBusy);

	IF  ton_TimeOut.Q THEN		// timeout
		int_TimeoutCounter[int_State]	:= int_TimeoutCounter[int_State]+1;
		fbShelly[int_State].bStart		:= FALSE;
		ton_TimeOut.IN 		:= FALSE;
		// go to next state
		IF 	int_state < 30 AND str_Array_IPs[int_State+1] <> '' THEN	
			int_State := int_State+1;
		ELSE
			int_State := 100;			// wait state for new run
		END_IF		
	ELSIF  fbShelly[int_State].bError THEN		// error
		int_ErrorCounter[int_State]	:= int_ErrorCounter[int_State]+1;
		fbShelly[int_State].bStart		:= FALSE;
		ton_TimeOut.IN 		:= FALSE;
		// go to next state
		IF 	int_state < 30 AND str_Array_IPs[int_State+1] <> '' THEN	
			int_State := int_State+1;
		ELSE
			int_State := 100;			// wait state for new run
		END_IF	
	ELSIF f_Trig_Busy[int_State].Q AND NOT fbShelly[int_State].bError AND NOT ton_TimeOut.Q THEN		// received values
		int_SuccessCounter[int_State]	:= int_SuccessCounter[int_State]+1;
		fbShelly[int_State].bStart		:= FALSE;
		ton_TimeOut.IN 		:= FALSE;
	
		
		// copy received values
		lrS5P1Voltage	:= fbShelly[int_State].lrvoltageP1; 
		lrS5P1Power 	:= fbShelly[int_State].lrpowerP1 * int_Multiplier_5;
		lrS5P1Energy 	:= fbShelly[int_State].lrenergyP1 *int_Multiplier_5;
		lrS5P1Temperature :=fbShelly[int_State].lrTemperatureP1;
		bS5P1Switch		:= fbShelly[int_State].bStateP1;
	

		// go to next state
		IF 	int_state < 30 AND str_Array_IPs[int_State+1] <> '' THEN	
			int_State :=int_State+1;
		ELSE
			int_State := 100;			// wait state for new run
		END_IF
	END_IF	
	
	6: 		// request
	
	fbShelly[int_State].bStart		:= TRUE;
	fbShelly[int_State].sHostname	:= str_Array_IPs[int_State];

	// values to transfer to shelly
	fbShelly[int_State].bOnP1		:= bS6P1On;
	fbShelly[int_State].bOffP1		:= bS6P1Off;
	
	ton_TimeOut.IN 		:= TRUE;
	f_Trig_Busy[int_State] (clk	:= fbShelly[int_State].bBusy);

	IF  ton_TimeOut.Q THEN		// timeout
		int_TimeoutCounter[int_State]	:= int_TimeoutCounter[int_State]+1;
		fbShelly[int_State].bStart		:= FALSE;
		ton_TimeOut.IN 		:= FALSE;
		// go to next state
		IF 	int_state < 30 AND str_Array_IPs[int_State+1] <> '' THEN	
			int_State := int_State+1;
		ELSE
			int_State := 100;			// wait state for new run
		END_IF		
	ELSIF  fbShelly[int_State].bError THEN		// error
		int_ErrorCounter[int_State]	:= int_ErrorCounter[int_State]+1;
		fbShelly[int_State].bStart		:= FALSE;
		ton_TimeOut.IN 		:= FALSE;
		// go to next state
		IF 	int_state < 30 AND str_Array_IPs[int_State+1] <> '' THEN	
			int_State := int_State+1;
		ELSE
			int_State := 100;			// wait state for new run
		END_IF	
	ELSIF f_Trig_Busy[int_State].Q AND NOT fbShelly[int_State].bError AND NOT ton_TimeOut.Q THEN		// received values
		int_SuccessCounter[int_State]	:= int_SuccessCounter[int_State]+1;
		fbShelly[int_State].bStart		:= FALSE;
		ton_TimeOut.IN 		:= FALSE;
	
		
		// copy received values
		lrS6P1Voltage	:= fbShelly[int_State].lrvoltageP1; 
		lrS6P1Power 	:= fbShelly[int_State].lrpowerP1 * int_Multiplier_6;
		lrS6P1Energy 	:= fbShelly[int_State].lrenergyP1 *int_Multiplier_6;
		lrS6P1Temperature :=fbShelly[int_State].lrTemperatureP1;
		bS6P1Switch		:= fbShelly[int_State].bStateP1;
	

		// go to next state
		IF 	int_state < 30 AND str_Array_IPs[int_State+1] <> '' THEN	
			int_State :=int_State+1;
		ELSE
			int_State := 100;			// wait state for new run
		END_IF
	END_IF	
	
	7: 		// request
	
	fbShelly[int_State].bStart		:= TRUE;
	fbShelly[int_State].sHostname	:= str_Array_IPs[int_State];

	// values to transfer to shelly
	fbShelly[int_State].bOnP1		:= bS7P1On;
	fbShelly[int_State].bOffP1		:= bS7P1Off;
	
	ton_TimeOut.IN 		:= TRUE;
	f_Trig_Busy[int_State] (clk	:= fbShelly[int_State].bBusy);

	IF  ton_TimeOut.Q THEN		// timeout
		int_TimeoutCounter[int_State]	:= int_TimeoutCounter[int_State]+1;
		fbShelly[int_State].bStart		:= FALSE;
		ton_TimeOut.IN 		:= FALSE;
		// go to next state
		IF 	int_state < 30 AND str_Array_IPs[int_State+1] <> '' THEN	
			int_State := int_State+1;
		ELSE
			int_State := 100;			// wait state for new run
		END_IF		
	ELSIF  fbShelly[int_State].bError THEN		// error
		int_ErrorCounter[int_State]	:= int_ErrorCounter[int_State]+1;
		fbShelly[int_State].bStart		:= FALSE;
		ton_TimeOut.IN 		:= FALSE;
		// go to next state
		IF 	int_state < 30 AND str_Array_IPs[int_State+1] <> '' THEN	
			int_State := int_State+1;
		ELSE
			int_State := 100;			// wait state for new run
		END_IF	
	ELSIF f_Trig_Busy[int_State].Q AND NOT fbShelly[int_State].bError AND NOT ton_TimeOut.Q THEN		// received values
		int_SuccessCounter[int_State]	:= int_SuccessCounter[int_State]+1;
		fbShelly[int_State].bStart		:= FALSE;
		ton_TimeOut.IN 		:= FALSE;
	
		
		// copy received values
		lrS7P1Voltage	:= fbShelly[int_State].lrvoltageP1; 
		lrS7P1Power 	:= fbShelly[int_State].lrpowerP1 * int_Multiplier_7;
		lrS7P1Energy 	:= fbShelly[int_State].lrenergyP1 *int_Multiplier_7;
		lrS7P1Temperature :=fbShelly[int_State].lrTemperatureP1;
		bS7P1Switch		:= fbShelly[int_State].bStateP1;
	

		// go to next state
		IF 	int_state < 30 AND str_Array_IPs[int_State+1] <> '' THEN	
			int_State :=int_State+1;
		ELSE
			int_State := 100;			// wait state for new run
		END_IF
	END_IF		

	8: 		// request
	
	fbShelly[int_State].bStart		:= TRUE;
	fbShelly[int_State].sHostname	:= str_Array_IPs[int_State];

	// values to transfer to shelly
	fbShelly[int_State].bOnP1		:= bS8P1On;
	fbShelly[int_State].bOffP1		:= bS8P1Off;
	
	ton_TimeOut.IN 		:= TRUE;
	f_Trig_Busy[int_State] (clk	:= fbShelly[int_State].bBusy);

	IF  ton_TimeOut.Q THEN		// timeout
		int_TimeoutCounter[int_State]	:= int_TimeoutCounter[int_State]+1;
		fbShelly[int_State].bStart		:= FALSE;
		ton_TimeOut.IN 		:= FALSE;
		// go to next state
		IF 	int_state < 30 AND str_Array_IPs[int_State+1] <> '' THEN	
			int_State := int_State+1;
		ELSE
			int_State := 100;			// wait state for new run
		END_IF		
	ELSIF  fbShelly[int_State].bError THEN		// error
		int_ErrorCounter[int_State]	:= int_ErrorCounter[int_State]+1;
		fbShelly[int_State].bStart		:= FALSE;
		ton_TimeOut.IN 		:= FALSE;
		// go to next state
		IF 	int_state < 30 AND str_Array_IPs[int_State+1] <> '' THEN	
			int_State := int_State+1;
		ELSE
			int_State := 100;			// wait state for new run
		END_IF	
	ELSIF f_Trig_Busy[int_State].Q AND NOT fbShelly[int_State].bError AND NOT ton_TimeOut.Q THEN		// received values
		int_SuccessCounter[int_State]	:= int_SuccessCounter[int_State]+1;
		fbShelly[int_State].bStart		:= FALSE;
		ton_TimeOut.IN 		:= FALSE;
	
		
		// copy received values
		lrS8P1Voltage	:= fbShelly[int_State].lrvoltageP1; 
		lrS8P1Power 	:= fbShelly[int_State].lrpowerP1 * int_Multiplier_8;
		lrS8P1Energy 	:= fbShelly[int_State].lrenergyP1 *int_Multiplier_8;
		lrS8P1Temperature :=fbShelly[int_State].lrTemperatureP1;
		bS8P1Switch		:= fbShelly[int_State].bStateP1;
	

		// go to next state
		IF 	int_state < 30 AND str_Array_IPs[int_State+1] <> '' THEN	
			int_State :=int_State+1;
		ELSE
			int_State := 100;			// wait state for new run
		END_IF
	END_IF	
	
	9: 		// request
	
	fbShelly[int_State].bStart		:= TRUE;
	fbShelly[int_State].sHostname	:= str_Array_IPs[int_State];

	// values to transfer to shelly
	fbShelly[int_State].bOnP1		:= bS9P1On;
	fbShelly[int_State].bOffP1		:= bS9P1Off;
	
	ton_TimeOut.IN 		:= TRUE;
	f_Trig_Busy[int_State] (clk	:= fbShelly[int_State].bBusy);

	IF  ton_TimeOut.Q THEN		// timeout
		int_TimeoutCounter[int_State]	:= int_TimeoutCounter[int_State]+1;
		fbShelly[int_State].bStart		:= FALSE;
		ton_TimeOut.IN 		:= FALSE;
		// go to next state
		IF 	int_state < 30 AND str_Array_IPs[int_State+1] <> '' THEN	
			int_State := int_State+1;
		ELSE
			int_State := 100;			// wait state for new run
		END_IF		
	ELSIF  fbShelly[int_State].bError THEN		// error
		int_ErrorCounter[int_State]	:= int_ErrorCounter[int_State]+1;
		fbShelly[int_State].bStart		:= FALSE;
		ton_TimeOut.IN 		:= FALSE;
		// go to next state
		IF 	int_state < 30 AND str_Array_IPs[int_State+1] <> '' THEN	
			int_State := int_State+1;
		ELSE
			int_State := 100;			// wait state for new run
		END_IF	
	ELSIF f_Trig_Busy[int_State].Q AND NOT fbShelly[int_State].bError AND NOT ton_TimeOut.Q THEN		// received values
		int_SuccessCounter[int_State]	:= int_SuccessCounter[int_State]+1;
		fbShelly[int_State].bStart		:= FALSE;
		ton_TimeOut.IN 		:= FALSE;
	
		
		// copy received values
		lrS9P1Voltage	:= fbShelly[int_State].lrvoltageP1; 
		lrS9P1Power 	:= fbShelly[int_State].lrpowerP1 * int_Multiplier_9;
		lrS9P1Energy 	:= fbShelly[int_State].lrenergyP1 *int_Multiplier_9;
		lrS9P1Temperature :=fbShelly[int_State].lrTemperatureP1;
		bS9P1Switch		:= fbShelly[int_State].bStateP1;
	

		// go to next state
		IF 	int_state < 30 AND str_Array_IPs[int_State+1] <> '' THEN	
				int_State :=int_State+1;

		ELSE
//			int_State :=int_State+2;													//										!!!!!!!!!!!!!!!!!!!!!!!!!!!!!!!!!!!!!!!!!!!!!!!!!!!!!!!!!!!!!!!!!!!!!!!!!!!!!!!!!!!!!!!!!!!!!!!!!!!!!!!!!!!!!!!!!!!!
			int_State := 100;			// wait state for new run
		END_IF
	END_IF		

	10: 		// request
	
	fbShelly[int_State].bStart		:= TRUE;
	fbShelly[int_State].sHostname	:= str_Array_IPs[int_State];

	// values to transfer to shelly
	fbShelly[int_State].bOnP1		:= bS10P1On;
	fbShelly[int_State].bOffP1		:= bS10P1Off;
	
	ton_TimeOut.IN 		:= TRUE;
	f_Trig_Busy[int_State] (clk	:= fbShelly[int_State].bBusy);

	IF  ton_TimeOut.Q THEN		// timeout
		int_TimeoutCounter[int_State]	:= int_TimeoutCounter[int_State]+1;
		fbShelly[int_State].bStart		:= FALSE;
		ton_TimeOut.IN 		:= FALSE;
		// go to next state
		IF 	int_state < 30 AND str_Array_IPs[int_State+1] <> '' THEN	
			int_State := int_State+1;
		ELSE
			int_State := 100;			// wait state for new run
		END_IF		
	ELSIF  fbShelly[int_State].bError THEN		// error
		int_ErrorCounter[int_State]	:= int_ErrorCounter[int_State]+1;
		fbShelly[int_State].bStart		:= FALSE;
		ton_TimeOut.IN 		:= FALSE;
		// go to next state
		IF 	int_state < 30 AND str_Array_IPs[int_State+1] <> '' THEN	
			int_State := int_State+1;
		ELSE
			int_State := 100;			// wait state for new run
		END_IF	
	ELSIF f_Trig_Busy[int_State].Q AND NOT fbShelly[int_State].bError AND NOT ton_TimeOut.Q THEN		// received values
		int_SuccessCounter[int_State]	:= int_SuccessCounter[int_State]+1;
		fbShelly[int_State].bStart		:= FALSE;
		ton_TimeOut.IN 		:= FALSE;
	
		
		// copy received values
		lrS10P1Voltage	:= fbShelly[int_State].lrvoltageP1; 
		lrS10P1Power 	:= fbShelly[int_State].lrpowerP1 * int_Multiplier_10;
		lrS10P1Energy 	:= fbShelly[int_State].lrenergyP1 *int_Multiplier_10;
		lrS10P1Temperature :=fbShelly[int_State].lrTemperatureP1;
		bS10P1Switch		:= fbShelly[int_State].bStateP1;
	

		// go to next state
		IF 	int_state < 30 AND str_Array_IPs[int_State+1] <> '' THEN	
			int_State :=int_State+1;
		ELSE
			int_State := 100;			// wait state for new run
		END_IF
	END_IF	

	11: 		// request
	
	fbShelly[int_State].bStart		:= TRUE;
	fbShelly[int_State].sHostname	:= str_Array_IPs[int_State];

	// values to transfer to shelly
	fbShelly[int_State].bOnP1		:= bS11P1On;
	fbShelly[int_State].bOffP1		:= bS11P1Off;
	
	ton_TimeOut.IN 		:= TRUE;
	f_Trig_Busy[int_State] (clk	:= fbShelly[int_State].bBusy);

	IF  ton_TimeOut.Q THEN		// timeout
		int_TimeoutCounter[int_State]	:= int_TimeoutCounter[int_State]+1;
		fbShelly[int_State].bStart		:= FALSE;
		ton_TimeOut.IN 		:= FALSE;
		// go to next state
		IF 	int_state < 30 AND str_Array_IPs[int_State+1] <> '' THEN	
			int_State := int_State+1;
		ELSE
			int_State := 100;			// wait state for new run
		END_IF		
	ELSIF  fbShelly[int_State].bError THEN		// error
		int_ErrorCounter[int_State]	:= int_ErrorCounter[int_State]+1;
		fbShelly[int_State].bStart		:= FALSE;
		ton_TimeOut.IN 		:= FALSE;
		// go to next state
		IF 	int_state < 30 AND str_Array_IPs[int_State+1] <> '' THEN	
			int_State := int_State+1;
		ELSE
			int_State := 100;			// wait state for new run
		END_IF	
	ELSIF f_Trig_Busy[int_State].Q AND NOT fbShelly[int_State].bError AND NOT ton_TimeOut.Q THEN		// received values
		int_SuccessCounter[int_State]	:= int_SuccessCounter[int_State]+1;
		fbShelly[int_State].bStart		:= FALSE;
		ton_TimeOut.IN 		:= FALSE;
	
		
		// copy received values
		lrS11P1Voltage	:= fbShelly[int_State].lrvoltageP1; 
		lrS11P1Power 	:= fbShelly[int_State].lrpowerP1 * int_Multiplier_11;
		lrS11P1Energy 	:= fbShelly[int_State].lrenergyP1 *int_Multiplier_11;
		lrS11P1Temperature :=fbShelly[int_State].lrTemperatureP1;
		bS11P1Switch	:= fbShelly[int_State].bStateP1;
		
		// go to next state
		IF 	int_state < 30 AND str_Array_IPs[int_State+1] <> '' THEN	
			int_State :=int_State+1;
		ELSE
			int_State := 100;			// wait state for new run
		END_IF
	END_IF
	
	12: 		// request
	
	fbShelly[int_State].bStart		:= TRUE;
	fbShelly[int_State].sHostname	:= str_Array_IPs[int_State];

	// values to transfer to shelly
	fbShelly[int_State].bOnP1		:= bS12P1On;
	fbShelly[int_State].bOffP1		:= bS12P1Off;
	
	ton_TimeOut.IN 		:= TRUE;
	f_Trig_Busy[int_State] (clk	:= fbShelly[int_State].bBusy);

	IF  ton_TimeOut.Q THEN		// timeout
		int_TimeoutCounter[int_State]	:= int_TimeoutCounter[int_State]+1;
		fbShelly[int_State].bStart		:= FALSE;
		ton_TimeOut.IN 		:= FALSE;
		// go to next state
		IF 	int_state < 30 AND str_Array_IPs[int_State+1] <> '' THEN	
			int_State := int_State+1;
		ELSE
			int_State := 100;			// wait state for new run
		END_IF		
	ELSIF  fbShelly[int_State].bError THEN		// error
		int_ErrorCounter[int_State]	:= int_ErrorCounter[int_State]+1;
		fbShelly[int_State].bStart		:= FALSE;
		ton_TimeOut.IN 		:= FALSE;
		// go to next state
		IF 	int_state < 30 AND str_Array_IPs[int_State+1] <> '' THEN	
			int_State := int_State+1;
		ELSE
			int_State := 100;			// wait state for new run
		END_IF	
	ELSIF f_Trig_Busy[int_State].Q AND NOT fbShelly[int_State].bError AND NOT ton_TimeOut.Q THEN		// received values
		int_SuccessCounter[int_State]	:= int_SuccessCounter[int_State]+1;
		fbShelly[int_State].bStart		:= FALSE;
		ton_TimeOut.IN 		:= FALSE;
	
		
		// copy received values
		lrS12P1Voltage	:= fbShelly[int_State].lrvoltageP1; 
		lrS12P1Power 	:= fbShelly[int_State].lrpowerP1 * int_Multiplier_12;
		lrS12P1Energy 	:= fbShelly[int_State].lrenergyP1 *int_Multiplier_12;
		lrS12P1Temperature :=fbShelly[int_State].lrTemperatureP1;
		bS12P1Switch		:= fbShelly[int_State].bStateP1;
		
		// go to next state
		IF 	int_state < 30 AND str_Array_IPs[int_State+1] <> '' THEN	
			int_State :=int_State+1;
		ELSE
			int_State := 100;			// wait state for new run
		END_IF
	END_IF

	13: 		// request
	
	fbShelly[int_State].bStart		:= TRUE;
	fbShelly[int_State].sHostname	:= str_Array_IPs[int_State];

	// values to transfer to shelly
	fbShelly[int_State].bOnP1		:= bS13P1On;
	fbShelly[int_State].bOffP1		:= bS13P1Off;
	
	ton_TimeOut.IN 		:= TRUE;
	f_Trig_Busy[int_State] (clk	:= fbShelly[int_State].bBusy);

	IF  ton_TimeOut.Q THEN		// timeout
		int_TimeoutCounter[int_State]	:= int_TimeoutCounter[int_State]+1;
		fbShelly[int_State].bStart		:= FALSE;
		ton_TimeOut.IN 		:= FALSE;
		// go to next state
		IF 	int_state < 30 AND str_Array_IPs[int_State+1] <> '' THEN	
			int_State := int_State+1;
		ELSE
			int_State := 100;			// wait state for new run
		END_IF		
	ELSIF  fbShelly[int_State].bError THEN		// error
		int_ErrorCounter[int_State]	:= int_ErrorCounter[int_State]+1;
		fbShelly[int_State].bStart		:= FALSE;
		ton_TimeOut.IN 		:= FALSE;
		// go to next state
		IF 	int_state < 30 AND str_Array_IPs[int_State+1] <> '' THEN	
			int_State := int_State+1;
		ELSE
			int_State := 100;			// wait state for new run
		END_IF	
	ELSIF f_Trig_Busy[int_State].Q AND NOT fbShelly[int_State].bError AND NOT ton_TimeOut.Q THEN		// received values
		int_SuccessCounter[int_State]	:= int_SuccessCounter[int_State]+1;
		fbShelly[int_State].bStart		:= FALSE;
		ton_TimeOut.IN 		:= FALSE;
	
		
		// copy received values
		lrS13P1Voltage	:= fbShelly[int_State].lrvoltageP1; 
		lrS13P1Power 	:= fbShelly[int_State].lrpowerP1 * int_Multiplier_13;
		lrS13P1Energy 	:= fbShelly[int_State].lrenergyP1 *int_Multiplier_13;
		lrS13P1Temperature :=fbShelly[int_State].lrTemperatureP1;
		bS13P1Switch	:= fbShelly[int_State].bStateP1;
		
		// go to next state
		IF 	int_state < 30 AND str_Array_IPs[int_State+1] <> '' THEN	
				int_State :=int_State+1;
		ELSE
//			int_State :=int_State+2;													//										!!!!!!!!!!!!!!!!!!!!!!!!!!!!!!!!!!!!!!!!!!!!!!!!!!!!!!!!!!!!!!!!!!!!!!!!!!!!!!!!!!!!!!!!!!!!!!!!!!!!!!!!!!!!!!!!!!!!
			int_State := 100;			// wait state for new run
		END_IF
	END_IF
	
	14: 		// request
	
	fbShelly[int_State].bStart		:= TRUE;
	fbShelly[int_State].sHostname	:= str_Array_IPs[int_State];

	// values to transfer to shelly
	fbShelly[int_State].bOnP1		:= bS14P1On;
	fbShelly[int_State].bOffP1		:= bS14P1Off;
	
	ton_TimeOut.IN 		:= TRUE;
	f_Trig_Busy[int_State] (clk	:= fbShelly[int_State].bBusy);

	IF  ton_TimeOut.Q THEN		// timeout
		int_TimeoutCounter[int_State]	:= int_TimeoutCounter[int_State]+1;
		fbShelly[int_State].bStart		:= FALSE;
		ton_TimeOut.IN 		:= FALSE;
		// go to next state
		IF 	int_state < 30 AND str_Array_IPs[int_State+1] <> '' THEN	
			int_State := int_State+1;
		ELSE
			int_State := 100;			// wait state for new run
		END_IF		
	ELSIF  fbShelly[int_State].bError THEN		// error
		int_ErrorCounter[int_State]	:= int_ErrorCounter[int_State]+1;
		fbShelly[int_State].bStart		:= FALSE;
		ton_TimeOut.IN 		:= FALSE;
		// go to next state
		IF 	int_state < 30 AND str_Array_IPs[int_State+1] <> '' THEN	
			int_State := int_State+1;
		ELSE
			int_State := 100;			// wait state for new run
		END_IF	
	ELSIF f_Trig_Busy[int_State].Q AND NOT fbShelly[int_State].bError AND NOT ton_TimeOut.Q THEN		// received values
		int_SuccessCounter[int_State]	:= int_SuccessCounter[int_State]+1;
		fbShelly[int_State].bStart		:= FALSE;
		ton_TimeOut.IN 		:= FALSE;
	
		
		// copy received values
		lrS14P1Voltage	:= fbShelly[int_State].lrvoltageP1; 
		lrS14P1Power 	:= fbShelly[int_State].lrpowerP1 * int_Multiplier_14;
		lrS14P1Energy 	:= fbShelly[int_State].lrenergyP1 *int_Multiplier_14;
		lrS14P1Temperature :=fbShelly[int_State].lrTemperatureP1;
		bS14P1Switch	:= fbShelly[int_State].bStateP1;
		
		// go to next state
		IF 	int_state < 30 AND str_Array_IPs[int_State+1] <> '' THEN	
			int_State :=int_State+1;
		ELSE
			int_State := 100;			// wait state for new run
		END_IF
	END_IF
		
	
	100:		// wait state
	ton_wait.IN :=TRUE;
	IF ton_wait.Q THEN
		ton_wait.IN :=FALSE;
		int_State := 1;
	END_IF
	
	
END_CASE

// Shelly communication

fbShelly[1](tDelayRequest:= T#0S, );
fbShelly[2](tDelayRequest:= T#0S, );
fbShelly[3](tDelayRequest:= T#0S, );
fbShelly[4](tDelayRequest:= T#0S, );
fbShelly[5](tDelayRequest:= T#0S, );
fbShelly[6](tDelayRequest:= T#0S, );
fbShelly[7](tDelayRequest:= T#0S, );
fbShelly[8](tDelayRequest:= T#0S, );
fbShelly[9](tDelayRequest:= T#0S, );
fbShelly[10](tDelayRequest:= T#0S, );
fbShelly[11](tDelayRequest:= T#0S, );
fbShelly[12](tDelayRequest:= T#0S, );
fbShelly[13](tDelayRequest:= T#0S, );
fbShelly[14](tDelayRequest:= T#0S, );

//timeout
ton_TimeOut(pt:=T#10S);

// wait
ton_wait(PT:=T#3S);
	

// re-calc to kW
lrS1P1Power_kW := lrS1P1Power / 1000;
lrS2P1Power_kW := lrS2P1Power / 1000;
lrS3P1Power_kW := lrS3P1Power / 1000;
lrS4P1Power_kW := lrS4P1Power / 1000;
lrS5P1Power_kW := lrS5P1Power / 1000;
lrS6P1Power_kW := lrS6P1Power / 1000;
lrS7P1Power_kW := lrS7P1Power / 1000;
lrS8P1Power_kW := lrS8P1Power / 1000;
lrS9P1Power_kW := lrS9P1Power / 1000;
lrS10P1Power_kW := lrS10P1Power / 1000;
lrS11P1Power_kW := lrS11P1Power / 1000;
lrS12P1Power_kW := lrS12P1Power / 1000;
lrS13P1Power_kW := lrS13P1Power / 1000;
lrS14P1Power_kW := lrS14P1Power / 1000;

// Other
lrRemainPower_kW := LIMIT(0, prg5530Grid.lrPowerGrid - (lrS1P1Power_kW + lrS2P1Power_kW + lrS3P1Power_kW + lrS4P1Power_kW + lrS5P1Power_kW + lrS6P1Power_kW + lrS7P1Power_kW + lrS8P1Power_kW + lrS9P1Power_kW + lrS10P1Power_kW + lrS11P1Power_kW + lrS12P1Power_kW + lrS13P1Power_kW + lrS14P1Power_kW), 999999);


// on / off commands from EMS

// AC Shelly 7
fbShelly[7].bEnableControl := TRUE;			// prg5530EMS.FB_TimeSwitch_AC.b_Enable;
IF prg5530EMS.FB_TimeSwitch_AC.b_Output_On AND NOT fbShelly[7].bStateP1 THEN
	bS7P1On :=TRUE;
ELSE
	bS7P1On := FALSE;
END_IF
IF NOT prg5530EMS.FB_TimeSwitch_AC.b_Output_On  AND fbShelly[7].bStateP1 THEN
	bS7P1Off :=TRUE;
ELSE
	bS7P1Off := FALSE;
END_IF
// Kondivitrione Shelly 6
fbShelly[6].bEnableControl := TRUE;			// prg5530EMS.FB_TimeSwitch_Vitrine.b_Enable;
IF prg5530EMS.FB_TimeSwitch_Vitrine.b_Output_On AND NOT fbShelly[6].bStateP1 THEN
	bS6P1On :=TRUE;
ELSE
	bS6P1On := FALSE;
END_IF
IF NOT prg5530EMS.FB_TimeSwitch_Vitrine.b_Output_On  AND fbShelly[6].bStateP1 THEN
	bS6P1Off :=TRUE;
ELSE
	bS6P1Off := FALSE;
END_IF
// Kühlmodul #1 (VK) Shelly 4 & Kühlmodul #3 (VK) Shelly 5 
fbShelly[4].bEnableControl := TRUE;			// prg5530EMS.FB_TimeSwitch_CoolingChamber.b_Enable;
IF prg5530EMS.FB_TimeSwitch_CoolingChamber.b_Output_On AND NOT fbShelly[4].bStateP1 THEN
	bS4P1On :=TRUE;
ELSE
	bS4P1On := FALSE;
END_IF
IF NOT prg5530EMS.FB_TimeSwitch_CoolingChamber.b_Output_On AND fbShelly[4].bStateP1 THEN
	bS4P1Off :=TRUE;
ELSE
	bS4P1Off := FALSE;
END_IF
fbShelly[5].bEnableControl := TRUE;			// prg5530EMS.FB_TimeSwitch_CoolingChamber.b_Enable;
IF prg5530EMS.FB_TimeSwitch_CoolingChamber.b_Output_On AND NOT fbShelly[5].bStateP1 THEN
	bS5P1On :=TRUE;
ELSE
	bS5P1On := FALSE;
END_IF
IF NOT prg5530EMS.FB_TimeSwitch_CoolingChamber.b_Output_On AND fbShelly[5].bStateP1 THEN
	bS5P1Off :=TRUE;
ELSE
	bS5P1Off := FALSE;
END_IF
// Boiler Shelly 12 + 13 + 14
fbShelly[12].bEnableControl := TRUE;			//  prg5530EMS.FB_TimeSwitch_Boiler.b_Enable;
IF prg5530EMS.FB_TimeSwitch_Boiler.b_Output_On AND NOT fbShelly[12].bStateP1 THEN
	bS12P1On :=TRUE;
ELSE
	bS12P1On := FALSE;
END_IF
IF NOT prg5530EMS.FB_TimeSwitch_Boiler.b_Output_On AND fbShelly[12].bStateP1 THEN
	bS12P1Off :=TRUE;
ELSE
	bS12P1Off := FALSE;
END_IF
fbShelly[13].bEnableControl := TRUE;			// prg5530EMS.FB_TimeSwitch_Boiler.b_Enable;
IF prg5530EMS.FB_TimeSwitch_Boiler.b_Output_On AND NOT fbShelly[13].bStateP1 THEN
	bS13P1On :=TRUE;
ELSE
	bS13P1On := FALSE;
END_IF
IF NOT prg5530EMS.FB_TimeSwitch_Boiler.b_Output_On AND fbShelly[13].bStateP1 THEN
	bS13P1Off :=TRUE;
ELSE
	bS13P1Off := FALSE;
END_IF
fbShelly[14].bEnableControl := TRUE;			// prg5530EMS.FB_TimeSwitch_Boiler.b_Enable;
IF prg5530EMS.FB_TimeSwitch_Boiler.b_Output_On AND NOT fbShelly[14].bStateP1 THEN
	bS14P1On :=TRUE;
ELSE
	bS14P1On := FALSE;
END_IF
IF NOT prg5530EMS.FB_TimeSwitch_Boiler.b_Output_On AND fbShelly[14].bStateP1 THEN
	bS14P1Off :=TRUE;
ELSE
	bS14P1Off := FALSE;
END_IF

// Außenbeleuchtung Shelly 11
fbShelly[11].bEnableControl := TRUE;			// prg5530EMS.FB_TimeSwitch_Outside.b_Enable;
IF prg5530EMS.RS_Outsidelight.Q1 AND NOT fbShelly[11].bStateP1 THEN
	bS11P1On :=TRUE;
ELSE
	bS11P1On := FALSE;
END_IF
IF NOT prg5530EMS.RS_Outsidelight.Q1 AND fbShelly[11].bStateP1 THEN
	bS11P1Off :=TRUE;
ELSE
	bS11P1Off := FALSE;
END_IF

// error bit to cloud 

m_Error_HTTP := fbShelly[4].bError OR fbShelly[5].bError OR fbShelly[6].bError OR fbShelly[7].bError OR fbShelly[11].bError OR fbShelly[12].bError OR fbShelly[13].bError OR fbShelly[14].bError;

END_PROGRAM

// ---- POUs/prg5530EMS.TcPOU
PROGRAM prg5530EMS
VAR
	bQ1Switch	AT%Q*	: BOOL;								//{#lynus.ag#()}

	FB_TimeSwitch_Coffee: FB_TimeSwitch_v2;
	FB_TimeSwitch_AC: FB_TimeSwitch_v2;				// Shelly 7
	FB_TimeSwitch_Vitrine: FB_TimeSwitch_v2;			// Shelly 6
	FB_TimeSwitch_CoolingChamber: FB_TimeSwitch_v2;	// Shelly 4 + 5
	FB_TimeSwitch_Outside: FB_TimeSwitch_v2;			// Shelly 11
	FB_TimeSwitch_Boiler: FB_TimeSwitch_v2;			// Shelly 12 + 13 + 14

	b_Coffee_Manual_On: BOOL;						//{#lynus.ag#()}
	b_Coffee_Manual_Off: BOOL;						//{#lynus.ag#()}
	b_AC_Manual_On: BOOL;							//{#lynus.ag#()}
	b_AC_Manual_Off: BOOL;							//{#lynus.ag#()}
	b_Vitrine_Manual_On: BOOL;						//{#lynus.ag#()}
	b_Vitrine_Manual_Off: BOOL;						//{#lynus.ag#()}
	b_CoolingChamber_Manual_On: BOOL;				//{#lynus.ag#()}
	b_CoolingChamber_Manual_Off: BOOL;				//{#lynus.ag#()}
	b_Outside_Manual_On: BOOL;						//{#lynus.ag#()}
	b_Outside_Manual_Off: BOOL;						//{#lynus.ag#()}
	b_Boiler_Manual_On: BOOL;						//{#lynus.ag#()}
	b_Boiler_Manual_Off: BOOL;						//{#lynus.ag#()}
	fbCalcSunriseSunset   		: FB_CalcSunriseSunset;
	todSunrise            		: TOD;
	todSunset             		: TOD;
	fb_GetTimeZoneInfo	:FB_GetTimeZoneInformation;
	b_firstCycle: BOOL;
	RS_Outsidelight: RS;
	r_trig_on: R_trig;
	r_trig_off: R_trig;
	b_Status_CoffeeMaschine: BOOL;					//{#lynus.ag#()}
	m_STart: BOOL;
END_VAR
VAR PERSISTENT
// opening hours
	byte_MoFr_Open_Hour		:BYTE;					//{#lynus.ag#()}
	byte_MoFr_Open_Minute	:BYTE;					//{#lynus.ag#()}
	byte_MoFr_Close_Hour	:BYTE;					//{#lynus.ag#()}
	byte_MoFr_Close_Minute	:BYTE;					//{#lynus.ag#()}
	byte_Sa_Open_Hour		:BYTE;					//{#lynus.ag#()}
	byte_Sa_Open_Minute		:BYTE;					//{#lynus.ag#()}
	byte_Sa_Close_Hour		:BYTE;					//{#lynus.ag#()}
	byte_Sa_Close_Minute	:BYTE;					//{#lynus.ag#()}
	byte_So_Open_Hour		:BYTE;					//{#lynus.ag#()}
	byte_So_Open_Minute		:BYTE;					//{#lynus.ag#()}
	byte_So_Close_Hour		:BYTE;					//{#lynus.ag#()}
	byte_So_Close_Minute	:BYTE;					//{#lynus.ag#()}
	
// offset coffeemaschine in hours			
	b_Enable_Control_Coffee		:BOOL;				//{#lynus.ag#()}
	real_Coffee_Offset_Start	:REAL;				//{#lynus.ag#()}
	real_Coffee_Offset_Stop		:REAL;				//{#lynus.ag#()}
// offset AC in hours			
	b_Enable_Control_AC			:BOOL;				//{#lynus.ag#()}
	real_AC_Offset_Start		:REAL;				//{#lynus.ag#()}
	real_AC_Offset_Stop			:REAL;				//{#lynus.ag#()}
// offset Vitrine in hours			
	b_Enable_Control_Vitrine	:BOOL;				//{#lynus.ag#()}
	real_Vitrine_Offset_Start	:REAL;				//{#lynus.ag#()}
	real_Vitrine_Offset_Stop	:REAL;				//{#lynus.ag#()}
// offset CoolingChamber in hours			
	b_Enable_Control_CoolingChamber	:BOOL;			//{#lynus.ag#()}
	real_CoolingChamber_Offset_Start :REAL;			//{#lynus.ag#()}
	real_CoolingChamber_Offset_Stop	:REAL;			//{#lynus.ag#()}
// offset Outside in hours			
	b_Enable_Control_Outside	:BOOL;				//{#lynus.ag#()}
	real_Outside_Offset_Start	:REAL;				//{#lynus.ag#()}
	real_Outside_Offset_Stop	:REAL;				//{#lynus.ag#()}
// offset Boiler in hours			
	b_Enable_Control_Boiler		:BOOL;				//{#lynus.ag#()}
	real_Boiler_Offset_Start	:REAL;				//{#lynus.ag#()}
	real_Boiler_Offset_Stop		:REAL;				//{#lynus.ag#()}
	
END_VAR

FB_TimeSwitch_Coffee(
	b_Enable:= b_Enable_Control_Coffee, 
	b_StatusOn:= NOT bQ1Switch, 
	structSystemTime:=prg_SystemTime.structSystemTime , 
	byte_MoFr_Open_Hour:= byte_MoFr_Open_Hour , 
	byte_MoFr_Open_Minute:= byte_MoFr_Open_Minute, 
	byte_MoFr_Close_Hour:= byte_MoFr_Close_Hour , 
	byte_MoFr_Close_Minute:= byte_MoFr_Close_Minute, 
	byte_Sa_Open_Hour:= byte_Sa_Open_Hour, 
	byte_Sa_Open_Minute:= byte_Sa_Open_Minute , 
	byte_Sa_Close_Hour:= byte_Sa_Close_Hour , 
	byte_Sa_Close_Minute:= byte_Sa_Close_Minute, 
	byte_So_Open_Hour:= byte_So_Open_Hour, 
	byte_So_Open_Minute:= byte_So_Open_Minute, 
	byte_So_Close_Hour:= byte_So_Close_Hour, 
	byte_So_Close_Minute:= byte_So_Close_Minute, 
	real_Offset_Start:= real_Coffee_Offset_Start , 
	real_Offset_Stop:= real_Coffee_Offset_Stop , 
	b_On_Manual:= b_Coffee_Manual_On, 
	b_Off_Manual:= b_Coffee_Manual_Off, 
	b_Output_On=> , 
	b_Error=> );
IF NOT FB_TimeSwitch_Coffee.b_Output_On THEN
	bQ1Switch := TRUE;
ELSIF FB_TimeSwitch_Coffee.b_Output_On THEN
	bQ1Switch := FALSE;
END_IF
b_Status_CoffeeMaschine := NOT bQ1Switch;

FB_TimeSwitch_AC(
	b_Enable:= b_Enable_Control_AC, 
	b_StatusOn:= prg5530CON.fbShelly[7].bStateP1, 
	structSystemTime:= prg_SystemTime.structSystemTime , 
	byte_MoFr_Open_Hour:= byte_MoFr_Open_Hour , 
	byte_MoFr_Open_Minute:= byte_MoFr_Open_Minute, 
	byte_MoFr_Close_Hour:= byte_MoFr_Close_Hour , 
	byte_MoFr_Close_Minute:= byte_MoFr_Close_Minute, 
	byte_Sa_Open_Hour:= byte_Sa_Open_Hour, 
	byte_Sa_Open_Minute:= byte_Sa_Open_Minute , 
	byte_Sa_Close_Hour:= byte_Sa_Close_Hour , 
	byte_Sa_Close_Minute:= byte_Sa_Close_Minute, 
	byte_So_Open_Hour:= byte_So_Open_Hour, 
	byte_So_Open_Minute:= byte_So_Open_Minute, 
	byte_So_Close_Hour:= byte_So_Close_Hour, 
	byte_So_Close_Minute:= byte_So_Close_Minute, 
	real_Offset_Start:= real_AC_Offset_Start , 
	real_Offset_Stop:= real_AC_Offset_Stop , 
	b_On_Manual:= b_AC_Manual_On, 
	b_Off_Manual:= b_AC_Manual_Off, 
	b_Output_On=> , 
	b_Error=> );

FB_TimeSwitch_Vitrine(
	b_Enable:= b_Enable_Control_Vitrine, 
	b_StatusOn:= prg5530CON.fbShelly[6].bStateP1, 
	structSystemTime:= prg_SystemTime.structSystemTime , 
	byte_MoFr_Open_Hour:= byte_MoFr_Open_Hour , 
	byte_MoFr_Open_Minute:= byte_MoFr_Open_Minute, 
	byte_MoFr_Close_Hour:= byte_MoFr_Close_Hour , 
	byte_MoFr_Close_Minute:= byte_MoFr_Close_Minute, 
	byte_Sa_Open_Hour:= byte_Sa_Open_Hour, 
	byte_Sa_Open_Minute:= byte_Sa_Open_Minute , 
	byte_Sa_Close_Hour:= byte_Sa_Close_Hour , 
	byte_Sa_Close_Minute:= byte_Sa_Close_Minute, 
	byte_So_Open_Hour:= byte_So_Open_Hour, 
	byte_So_Open_Minute:= byte_So_Open_Minute, 
	byte_So_Close_Hour:= byte_So_Close_Hour, 
	byte_So_Close_Minute:= byte_So_Close_Minute, 
	real_Offset_Start:= real_Vitrine_Offset_Start , 
	real_Offset_Stop:= real_Vitrine_Offset_Stop , 
	b_On_Manual:= b_Vitrine_Manual_On, 
	b_Off_Manual:= b_Vitrine_Manual_Off, 
	b_Output_On=> , 
	b_Error=> );

FB_TimeSwitch_CoolingChamber(
	b_Enable:= b_Enable_Control_CoolingChamber, 
	b_StatusOn:= prg5530CON.fbShelly[4].bStateP1 AND prg5530CON.fbShelly[5].bStateP1, 
	structSystemTime:= prg_SystemTime.structSystemTime , 
	byte_MoFr_Open_Hour:= byte_MoFr_Open_Hour , 
	byte_MoFr_Open_Minute:= byte_MoFr_Open_Minute, 
	byte_MoFr_Close_Hour:= byte_MoFr_Close_Hour , 
	byte_MoFr_Close_Minute:= byte_MoFr_Close_Minute, 
	byte_Sa_Open_Hour:= byte_Sa_Open_Hour, 
	byte_Sa_Open_Minute:= byte_Sa_Open_Minute , 
	byte_Sa_Close_Hour:= byte_Sa_Close_Hour , 
	byte_Sa_Close_Minute:= byte_Sa_Close_Minute, 
	byte_So_Open_Hour:= byte_So_Open_Hour, 
	byte_So_Open_Minute:= byte_So_Open_Minute, 
	byte_So_Close_Hour:= byte_So_Close_Hour, 
	byte_So_Close_Minute:= byte_So_Close_Minute, 
	real_Offset_Start:= real_CoolingChamber_Offset_Start , 
	real_Offset_Stop:= real_CoolingChamber_Offset_Stop , 
	b_On_Manual:= b_CoolingChamber_Manual_On, 
	b_Off_Manual:= b_CoolingChamber_Manual_Off, 
	b_Output_On=> , 
	b_Error=> );

FB_TimeSwitch_Outside(
	b_Enable:= b_Enable_Control_Outside, 
	b_StatusOn:= prg5530CON.fbShelly[11].bStateP1, 
	structSystemTime:= prg_SystemTime.structSystemTime , 
	byte_MoFr_Open_Hour:= byte_MoFr_Open_Hour , 
	byte_MoFr_Open_Minute:= byte_MoFr_Open_Minute, 
	byte_MoFr_Close_Hour:= byte_MoFr_Close_Hour , 
	byte_MoFr_Close_Minute:= byte_MoFr_Close_Minute, 
	byte_Sa_Open_Hour:= byte_Sa_Open_Hour, 
	byte_Sa_Open_Minute:= byte_Sa_Open_Minute , 
	byte_Sa_Close_Hour:= byte_Sa_Close_Hour , 
	byte_Sa_Close_Minute:= byte_Sa_Close_Minute, 
	byte_So_Open_Hour:= byte_So_Open_Hour, 
	byte_So_Open_Minute:= byte_So_Open_Minute, 
	byte_So_Close_Hour:= byte_So_Close_Hour, 
	byte_So_Close_Minute:= byte_So_Close_Minute, 
	real_Offset_Start:= real_Outside_Offset_Start , 
	real_Offset_Stop:= real_Outside_Offset_Stop , 
	b_On_Manual:= b_Outside_Manual_On, 
	b_Off_Manual:= b_Outside_Manual_Off, 
	b_Output_On=> , 
	b_Error=> );
	
// calculate sunset / sunrise
// find out the time details
fb_GetTimeZoneInfo(
	sNetID:= '', 
	bExecute:= prg_SystemTime.structSystemTime.wHour = 4 OR NOT b_firstCycle, 
	tTimeout:= T#5S, 
	bBusy=> , 
	bError=> , 
	nErrID=> , 
	tzID=> , 
	tzInfo=> );
b_firstCycle := TRUE;

fbCalcSunriseSunset(
	fDegreeOfLongitude := 16.3731,   (* Longitude of Vienna *)
	fDegreeOfLatitude := 48.2083,   (* Latitude of Vienna*)
	fReferenceMeridian := SEL( fb_GetTimeZoneInfo.tzID = eTimeZoneID_Daylight ,15,30),  (* Central European Time 15 Winter Timer / 30 Summer Time *)
	dCurrentDate := DT_TO_DATE(SYSTEMTIME_TO_Dt (prg_SystemTime.structSystemTime)),
	todSunrise => todSunrise,
	todSunset => todSunset);

r_trig_on (clk := FB_TimeSwitch_Outside.b_Output_On AND DT_TO_TOD(systemtime_to_dt(prg_SystemTime.structSystemTime))< (todSunrise +  T#1H) );
r_trig_off (clk := NOT FB_TimeSwitch_Outside.b_Output_On);

RS_Outsidelight(	Set := r_trig_on.Q OR ((todSunset - T#2H) =  DT_TO_TOD(systemtime_to_dt(prg_SystemTime.structSystemTime)) AND FB_TimeSwitch_Outside.b_Output_On) OR b_Outside_Manual_On ,
					Reset1 := r_trig_off.Q OR ((todSunrise +  T#1H)= DT_TO_TOD(systemtime_to_dt(prg_SystemTime.structSystemTime))) OR b_Outside_Manual_Off,
					Q1 => );	

FB_TimeSwitch_Boiler(
	b_Enable:= b_Enable_Control_Boiler, 
	b_StatusOn:= prg5530CON.fbShelly[12].bStateP1 AND prg5530CON.fbShelly[13].bStateP1 AND prg5530CON.fbShelly[14].bStateP1, 
	structSystemTime:= prg_SystemTime.structSystemTime , 
	byte_MoFr_Open_Hour:= byte_MoFr_Open_Hour , 
	byte_MoFr_Open_Minute:= byte_MoFr_Open_Minute, 
	byte_MoFr_Close_Hour:= byte_MoFr_Close_Hour , 
	byte_MoFr_Close_Minute:= byte_MoFr_Close_Minute, 
	byte_Sa_Open_Hour:= byte_Sa_Open_Hour, 
	byte_Sa_Open_Minute:= byte_Sa_Open_Minute , 
	byte_Sa_Close_Hour:= byte_Sa_Close_Hour , 
	byte_Sa_Close_Minute:= byte_Sa_Close_Minute, 
	byte_So_Open_Hour:= byte_So_Open_Hour, 
	byte_So_Open_Minute:= byte_So_Open_Minute, 
	byte_So_Close_Hour:= byte_So_Close_Hour, 
	byte_So_Close_Minute:= byte_So_Close_Minute, 
	real_Offset_Start:= real_Boiler_Offset_Start , 
	real_Offset_Stop:= real_Boiler_Offset_Stop , 
	b_On_Manual:= b_Boiler_Manual_On, 
	b_Off_Manual:= b_Boiler_Manual_Off, 
	b_Output_On=> , 
	b_Error=> );

END_PROGRAM

// ---- POUs/prgComEffIO.TcPOU
PROGRAM prgComEffIO
VAR
	fbCom		: FB_MqttCommunicator_V5;
END_VAR

fbCom(
	bConnect:= TRUE, 
	strAuthKey:=  'ENE87365342998' , 
	sUserName:= '7bc3790f-8cda-40cf-a3d0-fe533f4dbc31', 
	sUserPassword:= '3d47cfcf-7c65-4d9d-bca8-26b757b0fe92', 
	eSavePositionCertificate:= eSavePositionOnPLC.ePostionHardDisk, 
	time_HeartBeat_sec := T#1S,
	bConnected=> , 
	bError=> , 
	hrErrorCode=> , 
	eConnectionState=> , 
	eErrorMessage_Out=> );

END_PROGRAM
